ABB RAPID module: DrawRobotStudioCursive.mod

MODULE DrawRobotStudioCursive
  ! Hershey glyphs: FLo-ABB, MIT; see LICENSE-Hershey-ABB.txt.
  TASK PERS wobjdata wobjText := [FALSE,TRUE,"",[[370,-150,200],[1,0,0,0]],[[0,0,0],[1,0,0,0]]];
  CONST jointtarget jHome := [[0,0,0,0,30,0],[9E9,9E9,9E9,9E9,9E9,9E9]];
  CONST jointtarget jPhoto := [[150,0,0,0,30,0],[9E9,9E9,9E9,9E9,9E9,9E9]];
  VAR robtarget p;
  PERS num strokesDone := 0;
  PROC main()
    ConfL \Off;
    ConfJ \Off;
    Reset do_pen;
    strokesDone := 0;
    MoveAbsJ jHome,v100,fine,tool0;
    ! Stroke 1
    Point 0.00000,23.46479,10;
    MoveJ p,v100,fine,tool0\WObj:=wobjText;
    Point 0.00000,23.46479,0;
    MoveL p,v60,fine,tool0\WObj:=wobjText;
    Set do_pen;
    WaitTime 0.05;
    Point 2.76056,27.60563,0;
    MoveL p,v60,z0,tool0\WObj:=wobjText;
    Point 4.14085,30.36620,0;
    MoveL p,v60,z0,tool0\WObj:=wobjText;
    Point 4.14085,27.60563,0;
    MoveL p,v60,z0,tool0\WObj:=wobjText;
    Point 8.28169,27.60563,0;
    MoveL p,v60,z0,tool0\WObj:=wobjText;
    Point 9.66197,26.22535,0;
    MoveL p,v60,z0,tool0\WObj:=wobjText;
    Point 9.66197,23.46479,0;
    MoveL p,v60,z0,tool0\WObj:=wobjText;
    Point 8.28169,19.32394,0;
    MoveL p,v60,z0,tool0\WObj:=wobjText;
    Point 8.28169,17.94366,0;
    MoveL p,v60,z0,tool0\WObj:=wobjText;
    Point 9.66197,16.56338,0;
    MoveL p,v60,z0,tool0\WObj:=wobjText;
    Point 11.04225,16.56338,0;
    MoveL p,v60,z0,tool0\WObj:=wobjText;
    Point 13.80282,17.94366,0;
    MoveL p,v60,z0,tool0\WObj:=wobjText;
    Point 15.18310,19.32394,0;
    MoveL p,v60,z0,tool0\WObj:=wobjText;
    Point 17.94366,23.46479,0;
    MoveL p,v60,fine,tool0\WObj:=wobjText;
    Reset do_pen;
    WaitTime 0.05;
    Point 17.94366,23.46479,10;
    MoveL p,v60,fine,tool0\WObj:=wobjText;
    strokesDone := 1;
    ! Stroke 2
    Point 26.22535,28.98592,10;
    MoveJ p,v100,fine,tool0\WObj:=wobjText;
    Point 26.22535,28.98592,0;
    MoveL p,v60,fine,tool0\WObj:=wobjText;
    Set do_pen;
    WaitTime 0.05;
    Point 23.46479,28.98592,0;
    MoveL p,v60,z0,tool0\WObj:=wobjText;
    Point 20.70423,27.60563,0;
    MoveL p,v60,z0,tool0\WObj:=wobjText;
    Point 19.32394,26.22535,0;
    MoveL p,v60,z0,tool0\WObj:=wobjText;
    Point 17.94366,23.46479,0;
    MoveL p,v60,z0,tool0\WObj:=wobjText;
    Point 17.94366,20.70423,0;
    MoveL p,v60,z0,tool0\WObj:=wobjText;
    Point 19.32394,17.94366,0;
    MoveL p,v60,z0,tool0\WObj:=wobjText;
    Point 22.08451,16.56338,0;
    MoveL p,v60,z0,tool0\WObj:=wobjText;
    Point 24.84507,16.56338,0;
    MoveL p,v60,z0,tool0\WObj:=wobjText;
    Point 27.60563,17.94366,0;
    MoveL p,v60,z0,tool0\WObj:=wobjText;
    Point 28.98592,19.32394,0;
    MoveL p,v60,z0,tool0\WObj:=wobjText;
    Point 30.36620,22.08451,0;
    MoveL p,v60,z0,tool0\WObj:=wobjText;
    Point 30.36620,24.84507,0;
    MoveL p,v60,z0,tool0\WObj:=wobjText;
    Point 28.98592,27.60563,0;
    MoveL p,v60,z0,tool0\WObj:=wobjText;
    Point 26.22535,28.98592,0;
    MoveL p,v60,z0,tool0\WObj:=wobjText;
    Point 24.84507,27.60563,0;
    MoveL p,v60,z0,tool0\WObj:=wobjText;
    Point 24.84507,24.84507,0;
    MoveL p,v60,z0,tool0\WObj:=wobjText;
    Point 26.22535,22.08451,0;
    MoveL p,v60,z0,tool0\WObj:=wobjText;
    Point 28.98592,20.70423,0;
    MoveL p,v60,z0,tool0\WObj:=wobjText;
    Point 33.12676,20.70423,0;
    MoveL p,v60,z0,tool0\WObj:=wobjText;
    Point 35.88732,22.08451,0;
    MoveL p,v60,z0,tool0\WObj:=wobjText;
    Point 37.26761,23.46479,0;
    MoveL p,v60,fine,tool0\WObj:=wobjText;
    Reset do_pen;
    WaitTime 0.05;
    Point 37.26761,23.46479,10;
    MoveL p,v60,fine,tool0\WObj:=wobjText;
    strokesDone := 2;
    ! Stroke 3
    Point 37.26761,23.46479,10;
    MoveJ p,v100,fine,tool0\WObj:=wobjText;
    Point 37.26761,23.46479,0;
    MoveL p,v60,fine,tool0\WObj:=wobjText;
    Set do_pen;
    WaitTime 0.05;
    Point 40.02817,27.60563,0;
    MoveL p,v60,z0,tool0\WObj:=wobjText;
    Point 44.16901,34.50704,0;
    MoveL p,v60,z0,tool0\WObj:=wobjText;
    Point 45.54930,37.26761,0;
    MoveL p,v60,z0,tool0\WObj:=wobjText;
    Point 46.92958,41.40845,0;
    MoveL p,v60,z0,tool0\WObj:=wobjText;
    Point 46.92958,44.16901,0;
    MoveL p,v60,z0,tool0\WObj:=wobjText;
    Point 45.54930,45.54930,0;
    MoveL p,v60,z0,tool0\WObj:=wobjText;
    Point 42.78873,44.16901,0;
    MoveL p,v60,z0,tool0\WObj:=wobjText;
    Point 41.40845,41.40845,0;
    MoveL p,v60,z0,tool0\WObj:=wobjText;
    Point 40.02817,35.88732,0;
    MoveL p,v60,z0,tool0\WObj:=wobjText;
    Point 38.64789,26.22535,0;
    MoveL p,v60,z0,tool0\WObj:=wobjText;
    Point 38.64789,17.94366,0;
    MoveL p,v60,z0,tool0\WObj:=wobjText;
    Point 40.02817,16.56338,0;
    MoveL p,v60,z0,tool0\WObj:=wobjText;
    Point 41.40845,16.56338,0;
    MoveL p,v60,z0,tool0\WObj:=wobjText;
    Point 44.16901,17.94366,0;
    MoveL p,v60,z0,tool0\WObj:=wobjText;
    Point 46.92958,20.70423,0;
    MoveL p,v60,z0,tool0\WObj:=wobjText;
    Point 48.30986,24.84507,0;
    MoveL p,v60,z0,tool0\WObj:=wobjText;
    Point 48.30986,28.98592,0;
    MoveL p,v60,z0,tool0\WObj:=wobjText;
    Point 49.69014,23.46479,0;
    MoveL p,v60,z0,tool0\WObj:=wobjText;
    Point 51.07042,22.08451,0;
    MoveL p,v60,z0,tool0\WObj:=wobjText;
    Point 53.83099,22.08451,0;
    MoveL p,v60,z0,tool0\WObj:=wobjText;
    Point 56.59155,23.46479,0;
    MoveL p,v60,fine,tool0\WObj:=wobjText;
    Reset do_pen;
    WaitTime 0.05;
    Point 56.59155,23.46479,10;
    MoveL p,v60,fine,tool0\WObj:=wobjText;
    strokesDone := 3;
    ! Stroke 4
    Point 64.87324,28.98592,10;
    MoveJ p,v100,fine,tool0\WObj:=wobjText;
    Point 64.87324,28.98592,0;
    MoveL p,v60,fine,tool0\WObj:=wobjText;
    Set do_pen;
    WaitTime 0.05;
    Point 62.11268,28.98592,0;
    MoveL p,v60,z0,tool0\WObj:=wobjText;
    Point 59.35211,27.60563,0;
    MoveL p,v60,z0,tool0\WObj:=wobjText;
    Point 57.97183,26.22535,0;
    MoveL p,v60,z0,tool0\WObj:=wobjText;
    Point 56.59155,23.46479,0;
    MoveL p,v60,z0,tool0\WObj:=wobjText;
    Point 56.59155,20.70423,0;
    MoveL p,v60,z0,tool0\WObj:=wobjText;
    Point 57.97183,17.94366,0;
    MoveL p,v60,z0,tool0\WObj:=wobjText;
    Point 60.73239,16.56338,0;
    MoveL p,v60,z0,tool0\WObj:=wobjText;
    Point 63.49296,16.56338,0;
    MoveL p,v60,z0,tool0\WObj:=wobjText;
    Point 66.25352,17.94366,0;
    MoveL p,v60,z0,tool0\WObj:=wobjText;
    Point 67.63380,19.32394,0;
    MoveL p,v60,z0,tool0\WObj:=wobjText;
    Point 69.01408,22.08451,0;
    MoveL p,v60,z0,tool0\WObj:=wobjText;
    Point 69.01408,24.84507,0;
    MoveL p,v60,z0,tool0\WObj:=wobjText;
    Point 67.63380,27.60563,0;
    MoveL p,v60,z0,tool0\WObj:=wobjText;
    Point 64.87324,28.98592,0;
    MoveL p,v60,z0,tool0\WObj:=wobjText;
    Point 63.49296,27.60563,0;
    MoveL p,v60,z0,tool0\WObj:=wobjText;
    Point 63.49296,24.84507,0;
    MoveL p,v60,z0,tool0\WObj:=wobjText;
    Point 64.87324,22.08451,0;
    MoveL p,v60,z0,tool0\WObj:=wobjText;
    Point 67.63380,20.70423,0;
    MoveL p,v60,z0,tool0\WObj:=wobjText;
    Point 71.77465,20.70423,0;
    MoveL p,v60,z0,tool0\WObj:=wobjText;
    Point 74.53521,22.08451,0;
    MoveL p,v60,z0,tool0\WObj:=wobjText;
    Point 75.91549,23.46479,0;
    MoveL p,v60,fine,tool0\WObj:=wobjText;
    Reset do_pen;
    WaitTime 0.05;
    Point 75.91549,23.46479,10;
    MoveL p,v60,fine,tool0\WObj:=wobjText;
    strokesDone := 4;
    ! Stroke 5
    Point 75.91549,23.46479,10;
    MoveJ p,v100,fine,tool0\WObj:=wobjText;
    Point 75.91549,23.46479,0;
    MoveL p,v60,fine,tool0\WObj:=wobjText;
    Set do_pen;
    WaitTime 0.05;
    Point 78.67606,27.60563,0;
    MoveL p,v60,z0,tool0\WObj:=wobjText;
    Point 81.43662,33.12676,0;
    MoveL p,v60,fine,tool0\WObj:=wobjText;
    Reset do_pen;
    WaitTime 0.05;
    Point 81.43662,33.12676,10;
    MoveL p,v60,fine,tool0\WObj:=wobjText;
    strokesDone := 5;
    ! Stroke 6
    Point 85.57746,45.54930,10;
    MoveJ p,v100,fine,tool0\WObj:=wobjText;
    Point 85.57746,45.54930,0;
    MoveL p,v60,fine,tool0\WObj:=wobjText;
    Set do_pen;
    WaitTime 0.05;
    Point 77.29577,20.70423,0;
    MoveL p,v60,z0,tool0\WObj:=wobjText;
    Point 77.29577,17.94366,0;
    MoveL p,v60,z0,tool0\WObj:=wobjText;
    Point 78.67606,16.56338,0;
    MoveL p,v60,z0,tool0\WObj:=wobjText;
    Point 81.43662,16.56338,0;
    MoveL p,v60,z0,tool0\WObj:=wobjText;
    Point 84.19718,17.94366,0;
    MoveL p,v60,z0,tool0\WObj:=wobjText;
    Point 85.57746,19.32394,0;
    MoveL p,v60,z0,tool0\WObj:=wobjText;
    Point 88.33803,23.46479,0;
    MoveL p,v60,fine,tool0\WObj:=wobjText;
    Reset do_pen;
    WaitTime 0.05;
    Point 88.33803,23.46479,10;
    MoveL p,v60,fine,tool0\WObj:=wobjText;
    strokesDone := 6;
    ! Stroke 7
    Point 77.29577,34.50704,10;
    MoveJ p,v100,fine,tool0\WObj:=wobjText;
    Point 77.29577,34.50704,0;
    MoveL p,v60,fine,tool0\WObj:=wobjText;
    Set do_pen;
    WaitTime 0.05;
    Point 86.95775,34.50704,0;
    MoveL p,v60,fine,tool0\WObj:=wobjText;
    Reset do_pen;
    WaitTime 0.05;
    Point 86.95775,34.50704,10;
    MoveL p,v60,fine,tool0\WObj:=wobjText;
    strokesDone := 7;
    ! Stroke 8
    Point 88.33803,23.46479,10;
    MoveJ p,v100,fine,tool0\WObj:=wobjText;
    Point 88.33803,23.46479,0;
    MoveL p,v60,fine,tool0\WObj:=wobjText;
    Set do_pen;
    WaitTime 0.05;
    Point 91.09859,27.60563,0;
    MoveL p,v60,z0,tool0\WObj:=wobjText;
    Point 92.47887,30.36620,0;
    MoveL p,v60,z0,tool0\WObj:=wobjText;
    Point 92.47887,27.60563,0;
    MoveL p,v60,z0,tool0\WObj:=wobjText;
    Point 95.23944,23.46479,0;
    MoveL p,v60,z0,tool0\WObj:=wobjText;
    Point 96.61972,20.70423,0;
    MoveL p,v60,z0,tool0\WObj:=wobjText;
    Point 96.61972,17.94366,0;
    MoveL p,v60,z0,tool0\WObj:=wobjText;
    Point 93.85915,16.56338,0;
    MoveL p,v60,fine,tool0\WObj:=wobjText;
    Reset do_pen;
    WaitTime 0.05;
    Point 93.85915,16.56338,10;
    MoveL p,v60,fine,tool0\WObj:=wobjText;
    strokesDone := 8;
    ! Stroke 9
    Point 88.33803,17.94366,10;
    MoveJ p,v100,fine,tool0\WObj:=wobjText;
    Point 88.33803,17.94366,0;
    MoveL p,v60,fine,tool0\WObj:=wobjText;
    Set do_pen;
    WaitTime 0.05;
    Point 91.09859,16.56338,0;
    MoveL p,v60,z0,tool0\WObj:=wobjText;
    Point 96.61972,16.56338,0;
    MoveL p,v60,z0,tool0\WObj:=wobjText;
    Point 99.38028,17.94366,0;
    MoveL p,v60,z0,tool0\WObj:=wobjText;
    Point 100.76056,19.32394,0;
    MoveL p,v60,z0,tool0\WObj:=wobjText;
    Point 103.52113,23.46479,0;
    MoveL p,v60,fine,tool0\WObj:=wobjText;
    Reset do_pen;
    WaitTime 0.05;
    Point 103.52113,23.46479,10;
    MoveL p,v60,fine,tool0\WObj:=wobjText;
    strokesDone := 9;
    ! Stroke 10
    Point 103.52113,23.46479,10;
    MoveJ p,v100,fine,tool0\WObj:=wobjText;
    Point 103.52113,23.46479,0;
    MoveL p,v60,fine,tool0\WObj:=wobjText;
    Set do_pen;
    WaitTime 0.05;
    Point 106.28169,27.60563,0;
    MoveL p,v60,z0,tool0\WObj:=wobjText;
    Point 109.04225,33.12676,0;
    MoveL p,v60,fine,tool0\WObj:=wobjText;
    Reset do_pen;
    WaitTime 0.05;
    Point 109.04225,33.12676,10;
    MoveL p,v60,fine,tool0\WObj:=wobjText;
    strokesDone := 10;
    ! Stroke 11
    Point 113.18310,45.54930,10;
    MoveJ p,v100,fine,tool0\WObj:=wobjText;
    Point 113.18310,45.54930,0;
    MoveL p,v60,fine,tool0\WObj:=wobjText;
    Set do_pen;
    WaitTime 0.05;
    Point 104.90141,20.70423,0;
    MoveL p,v60,z0,tool0\WObj:=wobjText;
    Point 104.90141,17.94366,0;
    MoveL p,v60,z0,tool0\WObj:=wobjText;
    Point 106.28169,16.56338,0;
    MoveL p,v60,z0,tool0\WObj:=wobjText;
    Point 109.04225,16.56338,0;
    MoveL p,v60,z0,tool0\WObj:=wobjText;
    Point 111.80282,17.94366,0;
    MoveL p,v60,z0,tool0\WObj:=wobjText;
    Point 113.18310,19.32394,0;
    MoveL p,v60,z0,tool0\WObj:=wobjText;
    Point 115.94366,23.46479,0;
    MoveL p,v60,fine,tool0\WObj:=wobjText;
    Reset do_pen;
    WaitTime 0.05;
    Point 115.94366,23.46479,10;
    MoveL p,v60,fine,tool0\WObj:=wobjText;
    strokesDone := 11;
    ! Stroke 12
    Point 104.90141,34.50704,10;
    MoveJ p,v100,fine,tool0\WObj:=wobjText;
    Point 104.90141,34.50704,0;
    MoveL p,v60,fine,tool0\WObj:=wobjText;
    Set do_pen;
    WaitTime 0.05;
    Point 114.56338,34.50704,0;
    MoveL p,v60,fine,tool0\WObj:=wobjText;
    Reset do_pen;
    WaitTime 0.05;
    Point 114.56338,34.50704,10;
    MoveL p,v60,fine,tool0\WObj:=wobjText;
    strokesDone := 12;
    ! Stroke 13
    Point 115.94366,23.46479,10;
    MoveJ p,v100,fine,tool0\WObj:=wobjText;
    Point 115.94366,23.46479,0;
    MoveL p,v60,fine,tool0\WObj:=wobjText;
    Set do_pen;
    WaitTime 0.05;
    Point 118.70423,28.98592,0;
    MoveL p,v60,z0,tool0\WObj:=wobjText;
    Point 115.94366,20.70423,0;
    MoveL p,v60,z0,tool0\WObj:=wobjText;
    Point 115.94366,17.94366,0;
    MoveL p,v60,z0,tool0\WObj:=wobjText;
    Point 117.32394,16.56338,0;
    MoveL p,v60,z0,tool0\WObj:=wobjText;
    Point 120.08451,16.56338,0;
    MoveL p,v60,z0,tool0\WObj:=wobjText;
    Point 122.84507,17.94366,0;
    MoveL p,v60,z0,tool0\WObj:=wobjText;
    Point 125.60563,20.70423,0;
    MoveL p,v60,z0,tool0\WObj:=wobjText;
    Point 128.36620,24.84507,0;
    MoveL p,v60,fine,tool0\WObj:=wobjText;
    Reset do_pen;
    WaitTime 0.05;
    Point 128.36620,24.84507,10;
    MoveL p,v60,fine,tool0\WObj:=wobjText;
    strokesDone := 13;
    ! Stroke 14
    Point 129.74648,28.98592,10;
    MoveJ p,v100,fine,tool0\WObj:=wobjText;
    Point 129.74648,28.98592,0;
    MoveL p,v60,fine,tool0\WObj:=wobjText;
    Set do_pen;
    WaitTime 0.05;
    Point 126.98592,20.70423,0;
    MoveL p,v60,z0,tool0\WObj:=wobjText;
    Point 126.98592,17.94366,0;
    MoveL p,v60,z0,tool0\WObj:=wobjText;
    Point 128.36620,16.56338,0;
    MoveL p,v60,z0,tool0\WObj:=wobjText;
    Point 129.74648,16.56338,0;
    MoveL p,v60,z0,tool0\WObj:=wobjText;
    Point 132.50704,17.94366,0;
    MoveL p,v60,z0,tool0\WObj:=wobjText;
    Point 133.88732,19.32394,0;
    MoveL p,v60,z0,tool0\WObj:=wobjText;
    Point 136.64789,23.46479,0;
    MoveL p,v60,fine,tool0\WObj:=wobjText;
    Reset do_pen;
    WaitTime 0.05;
    Point 136.64789,23.46479,10;
    MoveL p,v60,fine,tool0\WObj:=wobjText;
    strokesDone := 14;
    ! Stroke 15
    Point 149.07042,24.84507,10;
    MoveJ p,v100,fine,tool0\WObj:=wobjText;
    Point 149.07042,24.84507,0;
    MoveL p,v60,fine,tool0\WObj:=wobjText;
    Set do_pen;
    WaitTime 0.05;
    Point 147.69014,27.60563,0;
    MoveL p,v60,z0,tool0\WObj:=wobjText;
    Point 144.92958,28.98592,0;
    MoveL p,v60,z0,tool0\WObj:=wobjText;
    Point 142.16901,28.98592,0;
    MoveL p,v60,z0,tool0\WObj:=wobjText;
    Point 139.40845,27.60563,0;
    MoveL p,v60,z0,tool0\WObj:=wobjText;
    Point 138.02817,26.22535,0;
    MoveL p,v60,z0,tool0\WObj:=wobjText;
    Point 136.64789,23.46479,0;
    MoveL p,v60,z0,tool0\WObj:=wobjText;
    Point 136.64789,20.70423,0;
    MoveL p,v60,z0,tool0\WObj:=wobjText;
    Point 138.02817,17.94366,0;
    MoveL p,v60,z0,tool0\WObj:=wobjText;
    Point 140.78873,16.56338,0;
    MoveL p,v60,z0,tool0\WObj:=wobjText;
    Point 143.54930,16.56338,0;
    MoveL p,v60,z0,tool0\WObj:=wobjText;
    Point 146.30986,17.94366,0;
    MoveL p,v60,z0,tool0\WObj:=wobjText;
    Point 147.69014,20.70423,0;
    MoveL p,v60,z0,tool0\WObj:=wobjText;
    Point 155.97183,45.54930,0;
    MoveL p,v60,fine,tool0\WObj:=wobjText;
    Reset do_pen;
    WaitTime 0.05;
    Point 155.97183,45.54930,10;
    MoveL p,v60,fine,tool0\WObj:=wobjText;
    strokesDone := 15;
    ! Stroke 16
    Point 150.45070,28.98592,10;
    MoveJ p,v100,fine,tool0\WObj:=wobjText;
    Point 150.45070,28.98592,0;
    MoveL p,v60,fine,tool0\WObj:=wobjText;
    Set do_pen;
    WaitTime 0.05;
    Point 149.07042,22.08451,0;
    MoveL p,v60,z0,tool0\WObj:=wobjText;
    Point 149.07042,17.94366,0;
    MoveL p,v60,z0,tool0\WObj:=wobjText;
    Point 150.45070,16.56338,0;
    MoveL p,v60,z0,tool0\WObj:=wobjText;
    Point 151.83099,16.56338,0;
    MoveL p,v60,z0,tool0\WObj:=wobjText;
    Point 154.59155,17.94366,0;
    MoveL p,v60,z0,tool0\WObj:=wobjText;
    Point 155.97183,19.32394,0;
    MoveL p,v60,z0,tool0\WObj:=wobjText;
    Point 158.73239,23.46479,0;
    MoveL p,v60,fine,tool0\WObj:=wobjText;
    Reset do_pen;
    WaitTime 0.05;
    Point 158.73239,23.46479,10;
    MoveL p,v60,fine,tool0\WObj:=wobjText;
    strokesDone := 16;
    ! Stroke 17
    Point 162.87324,35.88732,10;
    MoveJ p,v100,fine,tool0\WObj:=wobjText;
    Point 162.87324,35.88732,0;
    MoveL p,v60,fine,tool0\WObj:=wobjText;
    Set do_pen;
    WaitTime 0.05;
    Point 162.87324,34.50704,0;
    MoveL p,v60,z0,tool0\WObj:=wobjText;
    Point 164.25352,34.50704,0;
    MoveL p,v60,z0,tool0\WObj:=wobjText;
    Point 164.25352,35.88732,0;
    MoveL p,v60,z0,tool0\WObj:=wobjText;
    Point 162.87324,35.88732,0;
    MoveL p,v60,fine,tool0\WObj:=wobjText;
    Reset do_pen;
    WaitTime 0.05;
    Point 162.87324,35.88732,10;
    MoveL p,v60,fine,tool0\WObj:=wobjText;
    strokesDone := 17;
    ! Stroke 18
    Point 158.73239,23.46479,10;
    MoveJ p,v100,fine,tool0\WObj:=wobjText;
    Point 158.73239,23.46479,0;
    MoveL p,v60,fine,tool0\WObj:=wobjText;
    Set do_pen;
    WaitTime 0.05;
    Point 161.49296,28.98592,0;
    MoveL p,v60,z0,tool0\WObj:=wobjText;
    Point 158.73239,20.70423,0;
    MoveL p,v60,z0,tool0\WObj:=wobjText;
    Point 158.73239,17.94366,0;
    MoveL p,v60,z0,tool0\WObj:=wobjText;
    Point 160.11268,16.56338,0;
    MoveL p,v60,z0,tool0\WObj:=wobjText;
    Point 161.49296,16.56338,0;
    MoveL p,v60,z0,tool0\WObj:=wobjText;
    Point 164.25352,17.94366,0;
    MoveL p,v60,z0,tool0\WObj:=wobjText;
    Point 165.63380,19.32394,0;
    MoveL p,v60,z0,tool0\WObj:=wobjText;
    Point 168.39437,23.46479,0;
    MoveL p,v60,fine,tool0\WObj:=wobjText;
    Reset do_pen;
    WaitTime 0.05;
    Point 168.39437,23.46479,10;
    MoveL p,v60,fine,tool0\WObj:=wobjText;
    strokesDone := 18;
    ! Stroke 19
    Point 176.67606,28.98592,10;
    MoveJ p,v100,fine,tool0\WObj:=wobjText;
    Point 176.67606,28.98592,0;
    MoveL p,v60,fine,tool0\WObj:=wobjText;
    Set do_pen;
    WaitTime 0.05;
    Point 173.91549,28.98592,0;
    MoveL p,v60,z0,tool0\WObj:=wobjText;
    Point 171.15493,27.60563,0;
    MoveL p,v60,z0,tool0\WObj:=wobjText;
    Point 169.77465,26.22535,0;
    MoveL p,v60,z0,tool0\WObj:=wobjText;
    Point 168.39437,23.46479,0;
    MoveL p,v60,z0,tool0\WObj:=wobjText;
    Point 168.39437,20.70423,0;
    MoveL p,v60,z0,tool0\WObj:=wobjText;
    Point 169.77465,17.94366,0;
    MoveL p,v60,z0,tool0\WObj:=wobjText;
    Point 172.53521,16.56338,0;
    MoveL p,v60,z0,tool0\WObj:=wobjText;
    Point 175.29577,16.56338,0;
    MoveL p,v60,z0,tool0\WObj:=wobjText;
    Point 178.05634,17.94366,0;
    MoveL p,v60,z0,tool0\WObj:=wobjText;
    Point 179.43662,19.32394,0;
    MoveL p,v60,z0,tool0\WObj:=wobjText;
    Point 180.81690,22.08451,0;
    MoveL p,v60,z0,tool0\WObj:=wobjText;
    Point 180.81690,24.84507,0;
    MoveL p,v60,z0,tool0\WObj:=wobjText;
    Point 179.43662,27.60563,0;
    MoveL p,v60,z0,tool0\WObj:=wobjText;
    Point 176.67606,28.98592,0;
    MoveL p,v60,z0,tool0\WObj:=wobjText;
    Point 175.29577,27.60563,0;
    MoveL p,v60,z0,tool0\WObj:=wobjText;
    Point 175.29577,24.84507,0;
    MoveL p,v60,z0,tool0\WObj:=wobjText;
    Point 176.67606,22.08451,0;
    MoveL p,v60,z0,tool0\WObj:=wobjText;
    Point 179.43662,20.70423,0;
    MoveL p,v60,z0,tool0\WObj:=wobjText;
    Point 183.57746,20.70423,0;
    MoveL p,v60,z0,tool0\WObj:=wobjText;
    Point 186.33803,22.08451,0;
    MoveL p,v60,z0,tool0\WObj:=wobjText;
    Point 187.71831,23.46479,0;
    MoveL p,v60,fine,tool0\WObj:=wobjText;
    Reset do_pen;
    WaitTime 0.05;
    Point 187.71831,23.46479,10;
    MoveL p,v60,fine,tool0\WObj:=wobjText;
    strokesDone := 19;
    ! Stroke 20
    Point 193.23944,28.98592,10;
    MoveJ p,v100,fine,tool0\WObj:=wobjText;
    Point 193.23944,28.98592,0;
    MoveL p,v60,fine,tool0\WObj:=wobjText;
    Set do_pen;
    WaitTime 0.05;
    Point 218.08451,28.98592,0;
    MoveL p,v60,fine,tool0\WObj:=wobjText;
    Reset do_pen;
    WaitTime 0.05;
    Point 218.08451,28.98592,10;
    MoveL p,v60,fine,tool0\WObj:=wobjText;
    strokesDone := 20;
    ! Stroke 21
    Point 223.60563,23.46479,10;
    MoveJ p,v100,fine,tool0\WObj:=wobjText;
    Point 223.60563,23.46479,0;
    MoveL p,v60,fine,tool0\WObj:=wobjText;
    Set do_pen;
    WaitTime 0.05;
    Point 226.36620,27.60563,0;
    MoveL p,v60,z0,tool0\WObj:=wobjText;
    Point 229.12676,28.98592,0;
    MoveL p,v60,z0,tool0\WObj:=wobjText;
    Point 230.50704,27.60563,0;
    MoveL p,v60,z0,tool0\WObj:=wobjText;
    Point 230.50704,26.22535,0;
    MoveL p,v60,z0,tool0\WObj:=wobjText;
    Point 229.12676,20.70423,0;
    MoveL p,v60,z0,tool0\WObj:=wobjText;
    Point 227.74648,16.56338,0;
    MoveL p,v60,fine,tool0\WObj:=wobjText;
    Reset do_pen;
    WaitTime 0.05;
    Point 227.74648,16.56338,10;
    MoveL p,v60,fine,tool0\WObj:=wobjText;
    strokesDone := 21;
    ! Stroke 22
    Point 229.12676,20.70423,10;
    MoveJ p,v100,fine,tool0\WObj:=wobjText;
    Point 229.12676,20.70423,0;
    MoveL p,v60,fine,tool0\WObj:=wobjText;
    Set do_pen;
    WaitTime 0.05;
    Point 230.50704,23.46479,0;
    MoveL p,v60,z0,tool0\WObj:=wobjText;
    Point 233.26761,27.60563,0;
    MoveL p,v60,z0,tool0\WObj:=wobjText;
    Point 236.02817,28.98592,0;
    MoveL p,v60,z0,tool0\WObj:=wobjText;
    Point 238.78873,28.98592,0;
    MoveL p,v60,z0,tool0\WObj:=wobjText;
    Point 240.16901,27.60563,0;
    MoveL p,v60,z0,tool0\WObj:=wobjText;
    Point 240.16901,26.22535,0;
    MoveL p,v60,z0,tool0\WObj:=wobjText;
    Point 238.78873,20.70423,0;
    MoveL p,v60,z0,tool0\WObj:=wobjText;
    Point 237.40845,16.56338,0;
    MoveL p,v60,fine,tool0\WObj:=wobjText;
    Reset do_pen;
    WaitTime 0.05;
    Point 237.40845,16.56338,10;
    MoveL p,v60,fine,tool0\WObj:=wobjText;
    strokesDone := 22;
    ! Stroke 23
    Point 238.78873,20.70423,10;
    MoveJ p,v100,fine,tool0\WObj:=wobjText;
    Point 238.78873,20.70423,0;
    MoveL p,v60,fine,tool0\WObj:=wobjText;
    Set do_pen;
    WaitTime 0.05;
    Point 240.16901,23.46479,0;
    MoveL p,v60,z0,tool0\WObj:=wobjText;
    Point 242.92958,27.60563,0;
    MoveL p,v60,z0,tool0\WObj:=wobjText;
    Point 245.69014,28.98592,0;
    MoveL p,v60,z0,tool0\WObj:=wobjText;
    Point 248.45070,28.98592,0;
    MoveL p,v60,z0,tool0\WObj:=wobjText;
    Point 249.83099,27.60563,0;
    MoveL p,v60,z0,tool0\WObj:=wobjText;
    Point 249.83099,24.84507,0;
    MoveL p,v60,z0,tool0\WObj:=wobjText;
    Point 248.45070,20.70423,0;
    MoveL p,v60,z0,tool0\WObj:=wobjText;
    Point 248.45070,17.94366,0;
    MoveL p,v60,z0,tool0\WObj:=wobjText;
    Point 249.83099,16.56338,0;
    MoveL p,v60,z0,tool0\WObj:=wobjText;
    Point 251.21127,16.56338,0;
    MoveL p,v60,z0,tool0\WObj:=wobjText;
    Point 253.97183,17.94366,0;
    MoveL p,v60,z0,tool0\WObj:=wobjText;
    Point 255.35211,19.32394,0;
    MoveL p,v60,z0,tool0\WObj:=wobjText;
    Point 258.11268,23.46479,0;
    MoveL p,v60,fine,tool0\WObj:=wobjText;
    Reset do_pen;
    WaitTime 0.05;
    Point 258.11268,23.46479,10;
    MoveL p,v60,fine,tool0\WObj:=wobjText;
    strokesDone := 23;
    ! Stroke 24
    Point 267.77465,26.22535,10;
    MoveJ p,v100,fine,tool0\WObj:=wobjText;
    Point 267.77465,26.22535,0;
    MoveL p,v60,fine,tool0\WObj:=wobjText;
    Set do_pen;
    WaitTime 0.05;
    Point 267.77465,27.60563,0;
    MoveL p,v60,z0,tool0\WObj:=wobjText;
    Point 266.39437,28.98592,0;
    MoveL p,v60,z0,tool0\WObj:=wobjText;
    Point 263.63380,28.98592,0;
    MoveL p,v60,z0,tool0\WObj:=wobjText;
    Point 260.87324,27.60563,0;
    MoveL p,v60,z0,tool0\WObj:=wobjText;
    Point 259.49296,26.22535,0;
    MoveL p,v60,z0,tool0\WObj:=wobjText;
    Point 258.11268,23.46479,0;
    MoveL p,v60,z0,tool0\WObj:=wobjText;
    Point 258.11268,20.70423,0;
    MoveL p,v60,z0,tool0\WObj:=wobjText;
    Point 259.49296,17.94366,0;
    MoveL p,v60,z0,tool0\WObj:=wobjText;
    Point 262.25352,16.56338,0;
    MoveL p,v60,z0,tool0\WObj:=wobjText;
    Point 266.39437,16.56338,0;
    MoveL p,v60,z0,tool0\WObj:=wobjText;
    Point 270.53521,19.32394,0;
    MoveL p,v60,z0,tool0\WObj:=wobjText;
    Point 273.29577,23.46479,0;
    MoveL p,v60,fine,tool0\WObj:=wobjText;
    Reset do_pen;
    WaitTime 0.05;
    Point 273.29577,23.46479,10;
    MoveL p,v60,fine,tool0\WObj:=wobjText;
    strokesDone := 24;
    ! Stroke 25
    Point 273.29577,23.46479,10;
    MoveJ p,v100,fine,tool0\WObj:=wobjText;
    Point 273.29577,23.46479,0;
    MoveL p,v60,fine,tool0\WObj:=wobjText;
    Set do_pen;
    WaitTime 0.05;
    Point 276.05634,27.60563,0;
    MoveL p,v60,z0,tool0\WObj:=wobjText;
    Point 277.43662,30.36620,0;
    MoveL p,v60,z0,tool0\WObj:=wobjText;
    Point 276.05634,24.84507,0;
    MoveL p,v60,z0,tool0\WObj:=wobjText;
    Point 267.77465,0.00000,0;
    MoveL p,v60,fine,tool0\WObj:=wobjText;
    Reset do_pen;
    WaitTime 0.05;
    Point 267.77465,0.00000,10;
    MoveL p,v60,fine,tool0\WObj:=wobjText;
    strokesDone := 25;
    ! Stroke 26
    Point 276.05634,24.84507,10;
    MoveJ p,v100,fine,tool0\WObj:=wobjText;
    Point 276.05634,24.84507,0;
    MoveL p,v60,fine,tool0\WObj:=wobjText;
    Set do_pen;
    WaitTime 0.05;
    Point 277.43662,27.60563,0;
    MoveL p,v60,z0,tool0\WObj:=wobjText;
    Point 280.19718,28.98592,0;
    MoveL p,v60,z0,tool0\WObj:=wobjText;
    Point 282.95775,28.98592,0;
    MoveL p,v60,z0,tool0\WObj:=wobjText;
    Point 285.71831,27.60563,0;
    MoveL p,v60,z0,tool0\WObj:=wobjText;
    Point 287.09859,24.84507,0;
    MoveL p,v60,z0,tool0\WObj:=wobjText;
    Point 287.09859,22.08451,0;
    MoveL p,v60,z0,tool0\WObj:=wobjText;
    Point 285.71831,19.32394,0;
    MoveL p,v60,z0,tool0\WObj:=wobjText;
    Point 284.33803,17.94366,0;
    MoveL p,v60,z0,tool0\WObj:=wobjText;
    Point 281.57746,16.56338,0;
    MoveL p,v60,fine,tool0\WObj:=wobjText;
    Reset do_pen;
    WaitTime 0.05;
    Point 281.57746,16.56338,10;
    MoveL p,v60,fine,tool0\WObj:=wobjText;
    strokesDone := 26;
    ! Stroke 27
    Point 276.05634,17.94366,10;
    MoveJ p,v100,fine,tool0\WObj:=wobjText;
    Point 276.05634,17.94366,0;
    MoveL p,v60,fine,tool0\WObj:=wobjText;
    Set do_pen;
    WaitTime 0.05;
    Point 278.81690,16.56338,0;
    MoveL p,v60,z0,tool0\WObj:=wobjText;
    Point 282.95775,16.56338,0;
    MoveL p,v60,z0,tool0\WObj:=wobjText;
    Point 287.09859,17.94366,0;
    MoveL p,v60,z0,tool0\WObj:=wobjText;
    Point 289.85915,19.32394,0;
    MoveL p,v60,z0,tool0\WObj:=wobjText;
    Point 294.00000,23.46479,0;
    MoveL p,v60,fine,tool0\WObj:=wobjText;
    Reset do_pen;
    WaitTime 0.05;
    Point 294.00000,23.46479,10;
    MoveL p,v60,fine,tool0\WObj:=wobjText;
    strokesDone := 27;
    MoveAbsJ jHome,v100,fine,tool0;
    MoveAbsJ jPhoto,v100,fine,tool0;
  ERROR
    Reset do_pen;
    RAISE;
  ENDPROC
  PROC Point(num x,num y,num z)
    p := [[-y,x,z],[0,0,1,0],[0,0,0,0],[9E9,9E9,9E9,9E9,9E9,9E9]];
  ENDPROC
ENDMODULE
